(* CODESYS project Assembler_RECOVERED_2026-09-20T18-53-23.project

Project tree, tasks and I/O mapping:
  Device : CODESYS Control Win V3 x64, CODESYS, version 3.5.22.30
    application Application
      libraries: Standard, 3.5.22.0 (System)
      task MainTask (cyclic, interval t#20ms, priority 1) calls PLC_PRG
      program PLC_PRG [LD]
    Ethernet : Ethernet, CODESYS, version 4.2.0.0
      ModbusTCP_Server_Device : ModbusTCP Server Device, CODESYS, version 4.6.0.0
          settings: DistinctBitAreas = TRUE; Coils Size = 32; Discrete Inputs Size = 32
          output Application.PLC_PRG.CV1 : WORD  // Input Registers.Input Registers
          input  Application.PLC_PRG.Moving_x : BOOL  // Coils.Coils.Bit0
          input  Application.PLC_PRG.Moving_Z : BOOL  // Coils.Coils.Bit1
          input  Application.PLC_PRG.Sensor_item : BOOL  // Coils.Coils.Bit2
          input  Application.PLC_PRG.Sensor_Lid_atP : BOOL  // Coils.Coils.Bit3
          input  Application.PLC_PRG.Lim_Lid : BOOL  // Coils.Coils.Bit4
          input  Application.PLC_PRG.Sensor_Base_atP : BOOL  // Coils.Coils.Bit6
          input  Application.PLC_PRG.Part_Leave : BOOL  // Coils.Coils.Bit1
          input  Application.PLC_PRG.start : BOOL  // Coils.Coils.Bit2
          input  Application.PLC_PRG.Reset : BOOL  // Coils.Coils.Bit3
          input  Application.PLC_PRG.Stop : BOOL  // Coils.Coils.Bit4
          input  Application.PLC_PRG.E_Stop : BOOL  // Coils.Coils.Bit5
          input  Application.PLC_PRG.Stop_Grab : BOOL  // Coils.Coils.Bit6
          output Application.PLC_PRG.Move_x : BOOL  // Discrete Inputs.Discrete Inputs.Bit0
          output Application.PLC_PRG.Move_Z : BOOL  // Discrete Inputs.Discrete Inputs.Bit1
          output Application.PLC_PRG.Grab : BOOL  // Discrete Inputs.Discrete Inputs.Bit2
          output Application.PLC_PRG.lid_conv : BOOL  // Discrete Inputs.Discrete Inputs.Bit3
          output Application.PLC_PRG.Clamp_Lid : BOOL  // Discrete Inputs.Discrete Inputs.Bit4
          output Application.PLC_PRG.base_conv : BOOL  // Discrete Inputs.Discrete Inputs.Bit6
          output Application.PLC_PRG.Clamp_Base : BOOL  // Discrete Inputs.Discrete Inputs.Bit7
          output Application.PLC_PRG.Pos_Raise_B : BOOL  // Discrete Inputs.Discrete Inputs.Bit0
          unmapped channels: Holding Registers, Input Registers, Coils, Discrete Inputs
*)

// Device/Application/PLC_PRG
PROGRAM PLC_PRG
VAR
    (* --- BOOLEAN VARIABLES --- *)
    start: BOOL;
    Stop: BOOL;
    E_Stop: BOOL;
    Reset: BOOL;
    System_Running: BOOL;
    
    lid_conv: BOOL;
    base_conv: BOOL;
    Stop_Lid_Conv: BOOL;
    stop_conv_base: BOOL;
    
    Clamp_Lid: BOOL;
    Clamp_Base: BOOL;
    Pos_Raise_B: BOOL;
    
    Sensor_Lid_atP: BOOL;
    Sensor_Base_atP: BOOL;
    Sensor_item: BOOL;
    Lim_Lid: BOOL;
    Part_Leave: BOOL;
    Part_Cleared: BOOL;
    
    Move_x: BOOL;
    Moving_x: BOOL;
    Move_Z: BOOL;
    Moving_Z: BOOL;
    Arm_X_Return: BOOL;
    Arm_Z_Returned: BOOL;
    Arm_X_AtBase: BOOL;
    Lid_Placed: BOOL;
    
    Grab: BOOL;
    Stop_Grab: BOOL;
    Holding_Item: BOOL;

    (* --- TIMERS, COUNTERS & VALUES --- *)
    TOF_1: TOF;
    TOF_3: TOF;
    ET2: TIME;
    ET4: TIME;
    
    CTU_0: CTU;
    PV: WORD;
    CV1: WORD;

    (* --- TRIGGERS --- *)
    F_TRIG_0: F_TRIG;
    F_TRIG_1: F_TRIG;
    F_TRIG_2: F_TRIG;
    F_TRIG_3: F_TRIG;
    F_TRIG_4: F_TRIG;
    F_TRIG_5: F_TRIG;
	F_TRIG_6: F_TRIG;
    
    RS_0: RS;
    RS_1: RS;
    RS_2: RS;
    RS_3: RS;
    RS_4: RS;
    SR_5: SR;
	
END_VAR

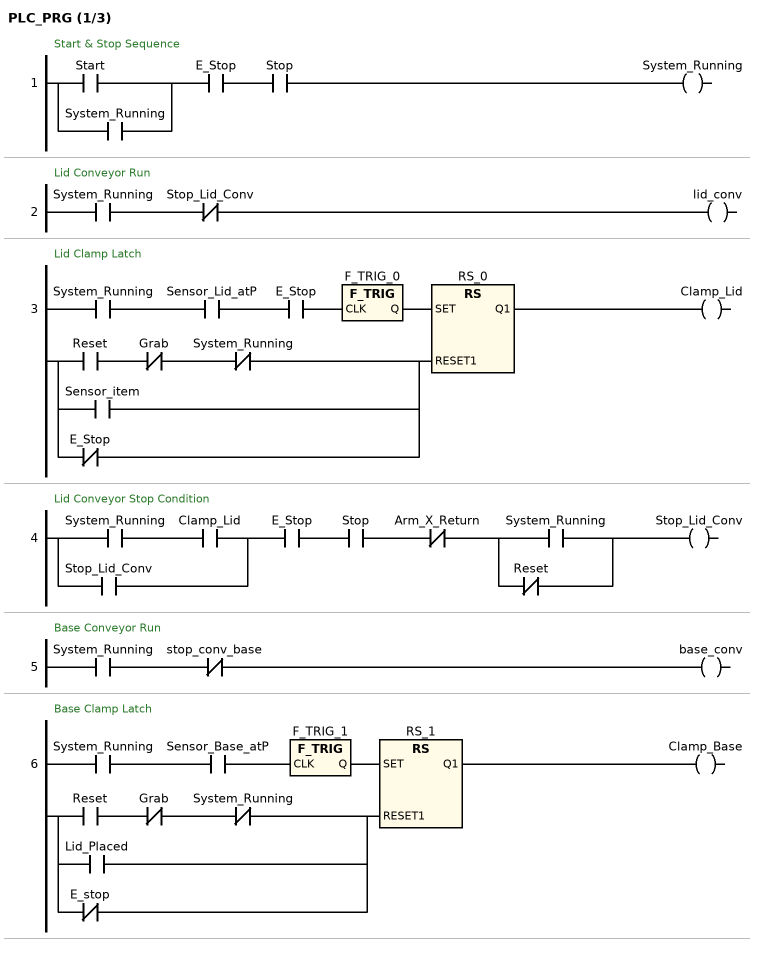
// NETWORK 1
// Start & Stop Sequence
System_Running := (Start OR System_Running) AND E_Stop AND Stop;

// NETWORK 2
// Lid Conveyor Run
lid_conv := System_Running AND NOT Stop_Lid_Conv;

// NETWORK 3
// Lid Clamp Latch
F_TRIG_0(CLK := System_Running AND Sensor_Lid_atP AND E_Stop); // F_TRIG
RS_0(SET := F_TRIG_0.Q, RESET1 := Reset AND NOT Grab AND NOT System_Running OR Sensor_item OR NOT E_Stop); // RS
Clamp_Lid := RS_0.Q1;

// NETWORK 4
// Lid Conveyor Stop Condition
Stop_Lid_Conv := (System_Running AND Clamp_Lid OR Stop_Lid_Conv) AND E_Stop AND Stop AND NOT Arm_X_Return AND (System_Running OR NOT Reset);

// NETWORK 5
// Base Conveyor Run
base_conv := System_Running AND NOT stop_conv_base;

// NETWORK 6
// Base Clamp Latch
F_TRIG_1(CLK := System_Running AND Sensor_Base_atP); // F_TRIG
RS_1(SET := F_TRIG_1.Q, RESET1 := Reset AND NOT Grab AND NOT System_Running OR Lid_Placed OR NOT E_stop); // RS
Clamp_Base := RS_1.Q1;

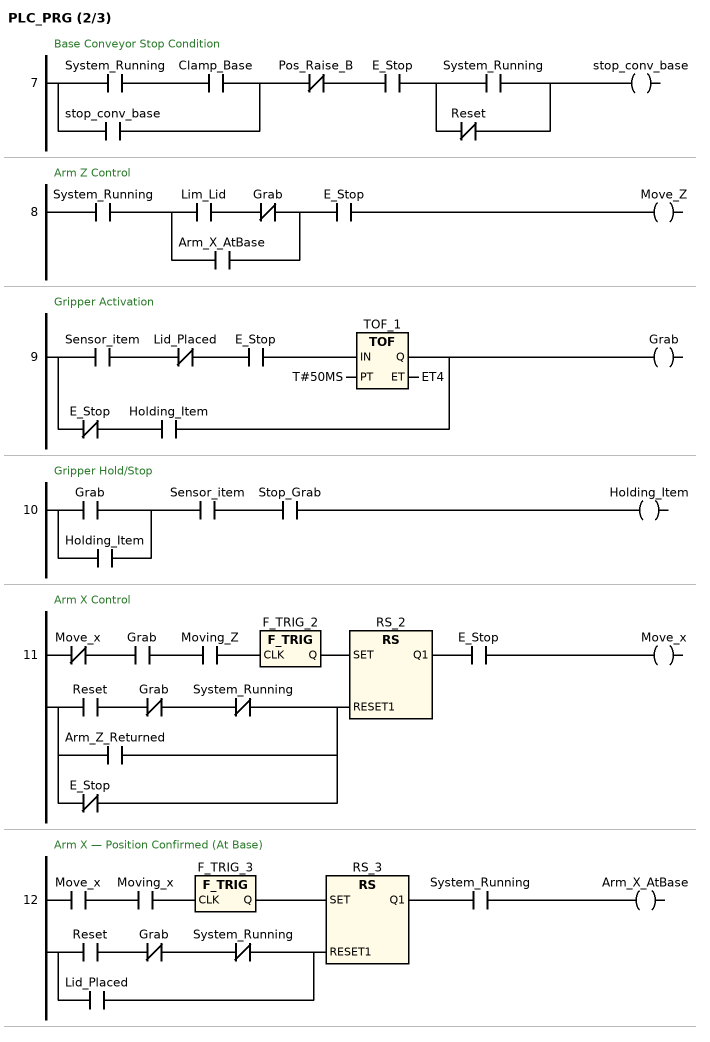
// NETWORK 7
// Base Conveyor Stop Condition
stop_conv_base := (System_Running AND Clamp_Base OR stop_conv_base) AND NOT Pos_Raise_B AND E_Stop AND (System_Running OR NOT Reset);

// NETWORK 8
// Arm Z Control
Move_Z := System_Running AND (Lim_Lid AND NOT Grab OR Arm_X_AtBase) AND E_Stop;

// NETWORK 9
// Gripper Activation
TOF_1(IN := Sensor_item AND NOT Lid_Placed AND E_Stop, PT := T#50MS, ET => ET4); // TOF
Grab := TOF_1.Q OR NOT E_Stop AND Holding_Item;

// NETWORK 10
// Gripper Hold/Stop
Holding_Item := (Grab OR Holding_Item) AND Sensor_item AND Stop_Grab;

// NETWORK 11
// Arm X Control
F_TRIG_2(CLK := NOT Move_x AND Grab AND Moving_Z); // F_TRIG
RS_2(SET := F_TRIG_2.Q, RESET1 := Reset AND NOT Grab AND NOT System_Running OR Arm_Z_Returned OR NOT E_Stop); // RS
Move_x := RS_2.Q1 AND E_Stop;

// NETWORK 12
// Arm X — Position Confirmed (At Base)
F_TRIG_3(CLK := Move_x AND Moving_x); // F_TRIG
RS_3(SET := F_TRIG_3.Q, RESET1 := Reset AND NOT Grab AND NOT System_Running OR Lid_Placed); // RS
Arm_X_AtBase := RS_3.Q1 AND System_Running;

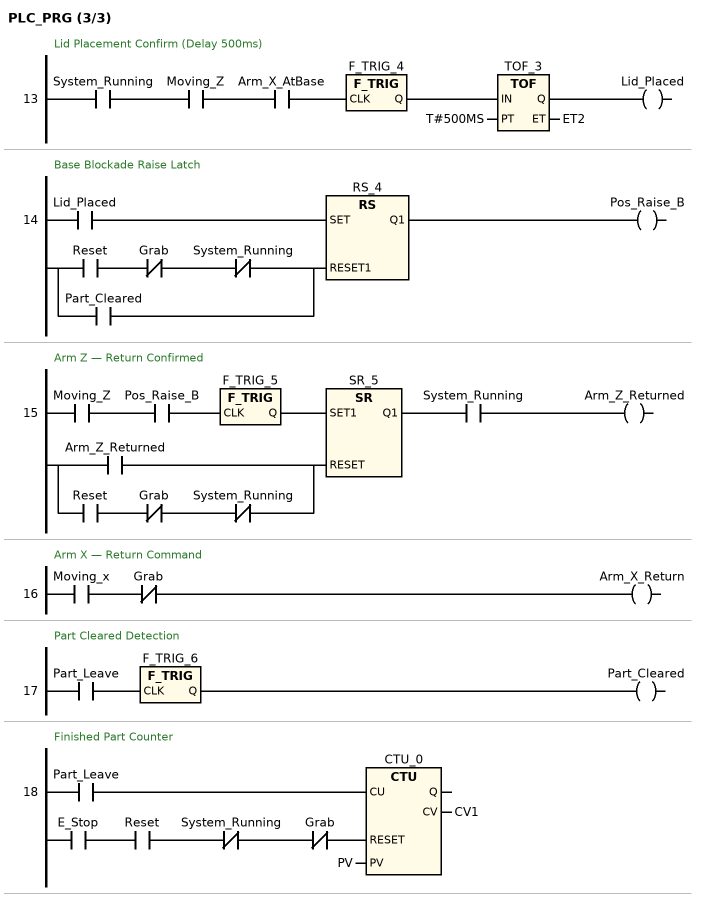
// NETWORK 13
// Lid Placement Confirm (Delay 500ms)
F_TRIG_4(CLK := System_Running AND Moving_Z AND Arm_X_AtBase); // F_TRIG
TOF_3(IN := F_TRIG_4.Q, PT := T#500MS, ET => ET2); // TOF
Lid_Placed := TOF_3.Q;

// NETWORK 14
// Base Blockade Raise Latch
RS_4(SET := Lid_Placed, RESET1 := Reset AND NOT Grab AND NOT System_Running OR Part_Cleared); // RS
Pos_Raise_B := RS_4.Q1;

// NETWORK 15
// Arm Z — Return Confirmed
F_TRIG_5(CLK := Moving_Z AND Pos_Raise_B); // F_TRIG
SR_5(SET1 := F_TRIG_5.Q, RESET := Arm_Z_Returned OR Reset AND NOT Grab AND NOT System_Running); // SR
Arm_Z_Returned := SR_5.Q1 AND System_Running;

// NETWORK 16
// Arm X — Return Command
Arm_X_Return := Moving_x AND NOT Grab;

// NETWORK 17
// Part Cleared Detection
F_TRIG_6(CLK := Part_Leave); // F_TRIG
Part_Cleared := F_TRIG_6.Q;

// NETWORK 18
// Finished Part Counter
CTU_0(CU := Part_Leave, RESET := E_Stop AND Reset AND NOT System_Running AND NOT Grab, PV := PV, CV => CV1); // CTU

END_PROGRAM
